FUNCTION_BLOCK FB_SUNPOS
VAR_INPUT
	// Julian Date
	JD:		LREAL;
	// output in Radians instead of Degrees
	RADIAN:	BOOL:= FALSE;
END_VAR
VAR_OUTPUT
	RA,
	Dec,
	longmed,
	oblt:	LREAL;
END_VAR
VAR
	t, //  Julian centuries FROM 1900.0
	l, //  sun's mean longitude
	me, // Earth's mean anomaly
	ellcor, // ellipticity of the orbit
	mv, // mean anomaly of Venus
	vencorr,
	mm, 
	marscorr,
mj, jupcorr,
d, longterm, mooncorr,  omega:	LREAL;
END_VAR
VAR CONSTANT
	dtor: LREAL := PI/180.0; // Pi/180
END_VAR

(* source: https://idlastro.gsfc.nasa.gov/ftp/pro/astro/sunpos.pro *)

//  form TIME in Julian centuries FROM 1900.0
t := (jd - 2415020.0)/36525.0;

//  form sun's mean longitude
l := (279.696678+LMOD(36000.768925*t, 360.0))*3600.0;

//  allow for ellipticity of the orbit (equation of centre) using the Earth's mean anomaly ME
me := 358.475844 + LMOD(35999.049750*t, 360.0);
ellcor  := (6910.1 - 17.2*t)*SIN(me*dtor) + 72.3*SIN(2.0*me*dtor);
l := l + ellcor;
 
// allow FOR the Venus perturbations using the mean anomaly OF Venus MV
mv := 212.603219 + LMOD(58517.803875*t, 360.0);
vencorr := 4.8 * COS((299.1017 + mv - me)*dtor) + 
          5.5 * COS((148.3133 +  2.0 * mv  -  2.0 * me )*dtor) + 
          2.5 * COS((315.9433 +  2.0 * mv  -  3.0 * me )*dtor) + 
          1.6 * COS((345.2533 +  3.0 * mv  -  4.0 * me )*dtor) + 
          1.0 * COS((318.15   +  3.0 * mv  -  5.0 * me )*dtor);
l := l + vencorr;

//  Allow FOR the Mars perturbations using the mean anomaly OF Mars MM
mm := 319.529425  +  LMOD( 19139.858500 * t,  360.0 );
marscorr := 2.0 * COS((343.8883 -  2.0 * mm  +  2.0 * me)*dtor ) + 
            1.8 * COS((200.4017 -  2.0 * mm  + me) * dtor);
l := l + marscorr;

// Allow FOR the Jupiter perturbations using the mean anomaly OF Jupiter MJ
mj := 225.328328  +  LMOD( 3034.6920239 * t,  360.0 );
jupcorr := 7.2 * COS(( 179.5317 - mj + me )*dtor) + 
          2.6 * COS((263.2167  -  MJ ) *dtor) + 
          2.7 * COS(( 87.1450  -  2.0 * mj  +  2.0 * me ) *dtor) + 
          1.6 * COS((109.4933  -  2.0 * mj  +  me ) *dtor);
l := l + jupcorr;

// Allow FOR the Moons perturbations using the mean elongation OF the Moon from the Sun D
d := 350.7376814  + LMOD( 445267.11422 * t,  360.0 );
mooncorr  := 6.5 * SIN(d*dtor);
l := l + mooncorr;

// Allow for long period terms
longterm := 6.4 * SIN(( 231.19  +  20.20 * t )*dtor);
l :=  l + longterm;
l :=  LMOD( l + 2592000.0,  1296000.0); 
longmed := l/3600.0;

// Allow for Aberration
l :=  l - 20.5;

// Allow for Nutation using the longitude of the Moons mean node OMEGA
omega := 259.183275 - LMOD( 1934.142008 * t, 360.0);
l :=  l - 17.2 * SIN(omega*dtor);

// Form the True Obliquity
oblt := 23.452294 - 0.0130125*t + (9.2*COS(omega*dtor))/3600.0;

// Form Right Ascension AND Declination
l := l/3600.0;
ra := ATAN2( SIN(l*dtor) * COS(oblt*dtor), COS(l*dtor) );
ra := MODABS(ra, 360.0);
dec := ASIN(SIN(l*dtor) * SIN(oblt*dtor));
 
IF RADIAN THEN
	oblt := oblt*dtor; 
	longmed := longmed*dtor;
ELSE
	ra := ra/dtor;
    dec := dec/dtor;
END_IF

END_FUNCTION_BLOCK

(* stored: Version 1.1.0.1, ProductVersion 3.1.4022.17
   POU FB_SUNPOS: Id {0dff82b7-3e2e-4cb4-82b3-58dc17eb6623}, SpecialFunc None *)
